FUNCTION_BLOCK FB_Bel_Taster_Steuerung
VAR_INPUT
END_VAR
VAR_OUTPUT
	Betrieb			: BOOL:=TRUE;
	BIN				: BOOL;
	auto_Modus		: BOOL;
END_VAR
VAR
	IN_Bin	AT %I* : BOOL;

	Taster			: R_TRIG;
	Halter			: RS;
	Licht_Schalten	: SINT := 2;

	Taster_Virtuell	: TP;
	Warte_Zeit		:TON;
	Halter1			: RS;
	Taste			: BOOL:=TRUE;	(*verstaerkung steigen*)
	Taste2			: BOOL;			(*nach 4s TRUE auto_Modus einsetzen*)
END_VAR
VAR // added by the converter: edge detectors and wires of the graphical bodies
    _w1, _w2, _w3, _w5 : ANY;
    _w4, _w6 : BOOL;
END_VAR

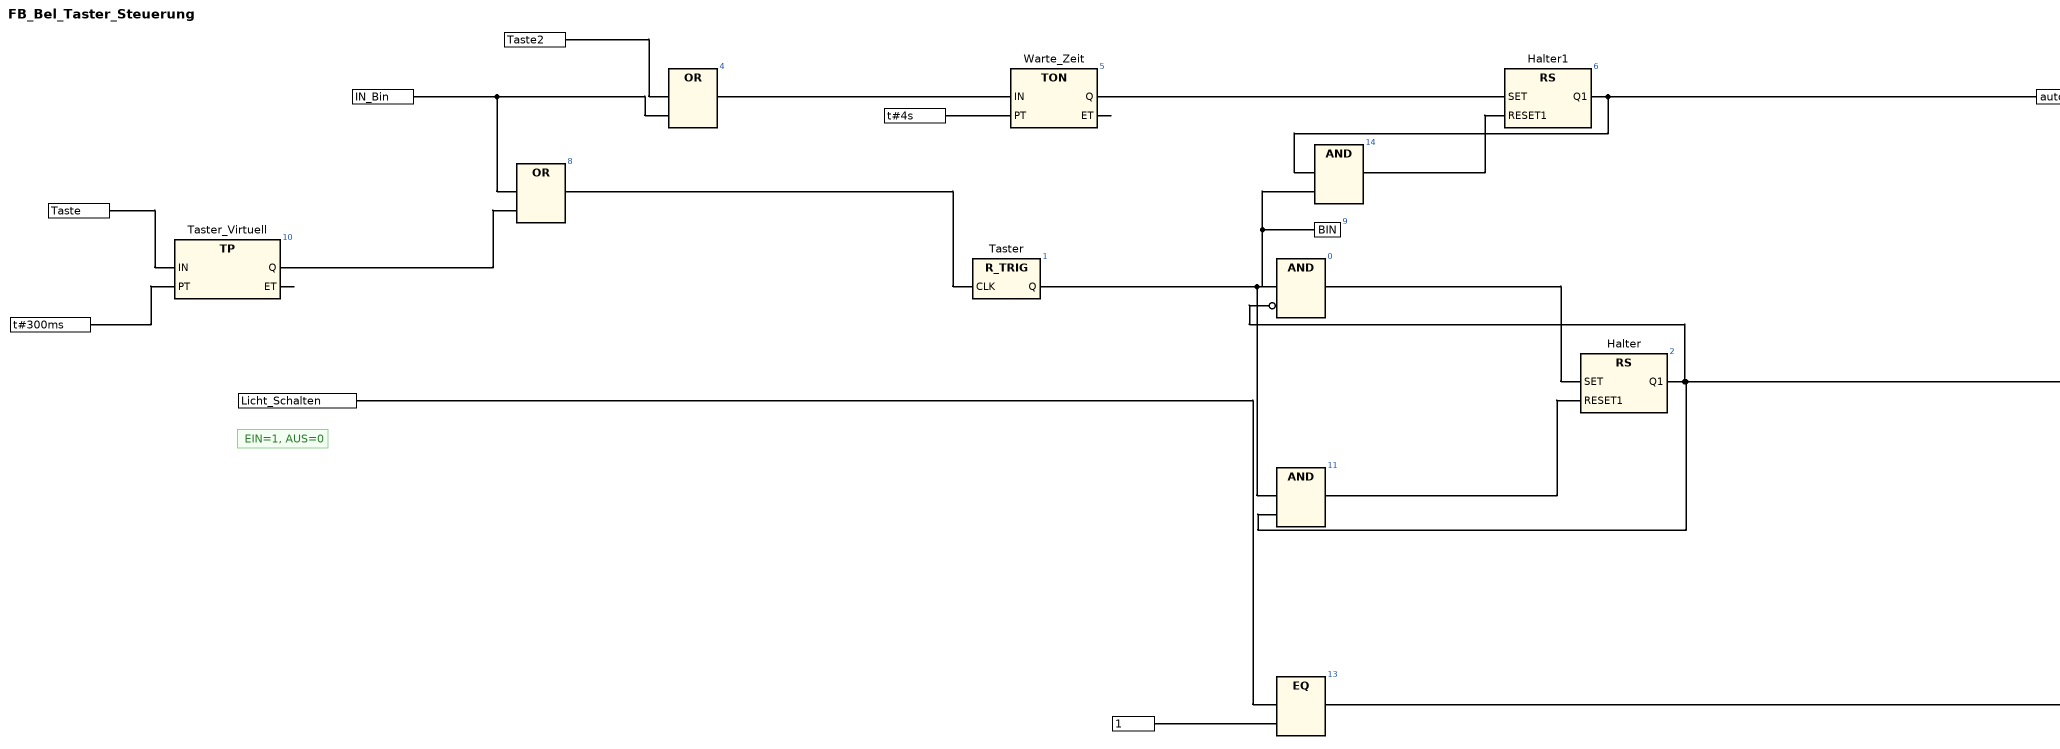
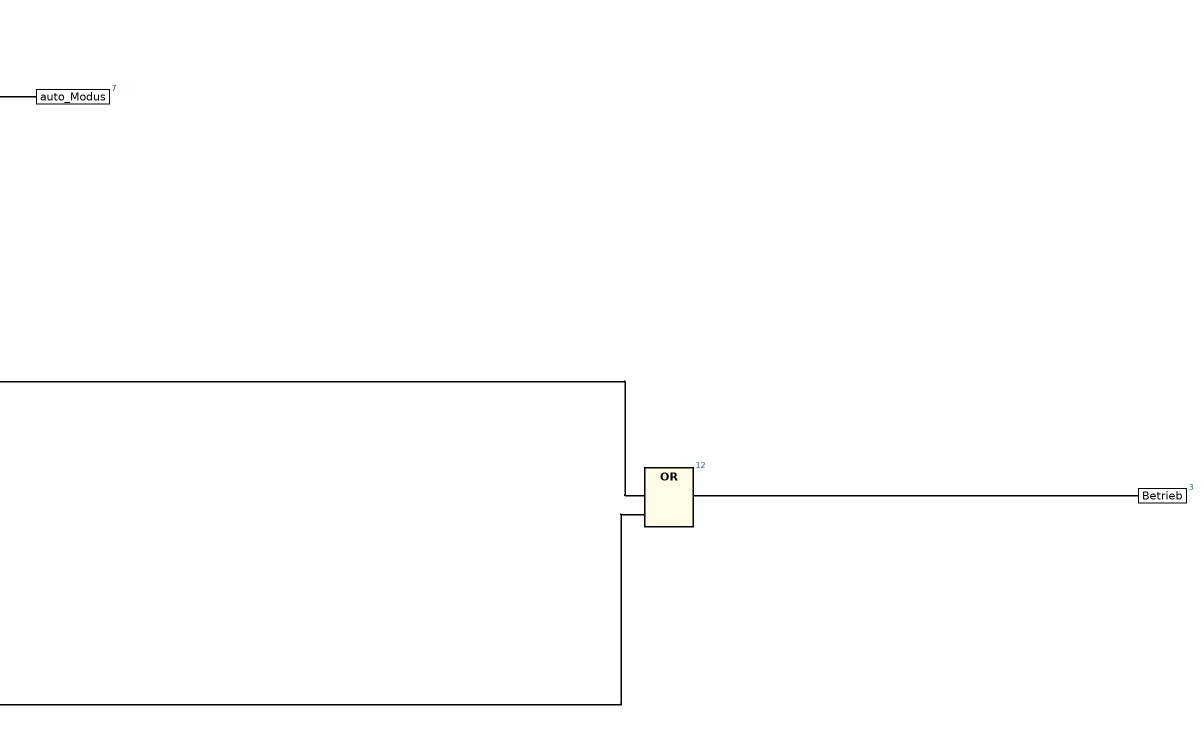
_w1 := Taster.Q AND NOT Halter.Q1;
Taster(CLK := _w2); // R_TRIG
Halter(SET := _w1, RESET1 := _w3); // RS
Betrieb := _w4;
Warte_Zeit(IN := Taste2 OR IN_Bin, PT := t#4s); // TON
Halter1(SET := Warte_Zeit.Q, RESET1 := _w5); // RS
auto_Modus := Halter1.Q1;
_w2 := IN_Bin OR Taster_Virtuell.Q;
BIN := Taster.Q;
Taster_Virtuell(IN := Taste, PT := t#300ms); // TP
//  EIN=1, AUS=0
_w3 := Taster.Q AND Halter.Q1;
_w4 := Halter.Q1 OR _w6;
_w6 := Licht_Schalten = 1;
_w5 := Halter1.Q1 AND Taster.Q;

END_FUNCTION_BLOCK

(* stored: Version 1.1.0.1, ProductVersion 3.1.4024.9
   POU FB_Bel_Taster_Steuerung: Id {9cdffb90-46f2-49ed-9b32-750ad19cefc4}, SpecialFunc None *)
